FUNCTION_BLOCK VirtualMaster EXTENDS FB_PackML_BaseModule
VAR
	Axis : FB_Component_BasicSlaveAxis := (Name := 'Virtual Master');
END_VAR

METHOD PROTECTED Aborting
//Mode is ignored
CASE SequenceState OF
	0:
		NoStateTasksToComplete := FALSE;

		// Stop Axis
		Axis.Override := 100;
		IF Axis.Stop() OR Axis.Error THEN // This will also GearOut
			SequenceState := SequenceState + 10;
		END_IF

	10:
		IF Axis.Stopped THEN
			SequenceState := SequenceState + 10;
		END_IF

	20: // Disable Axis
		IF Axis.Disable() THEN
			SequenceState := SequenceState + 10;
		END_IF

	30:
		IF NOT Axis.Enabled THEN
			SequenceState := SequenceState + 10;
		END_IF

	40:
		StateTasksComplete := TRUE;
END_CASE

SUPER^.Aborting();
END_METHOD

PROPERTY AxisRef : REFERENCE TO AXIS_REF
GET
AxisRef REF= Axis.Axis;
END_GET
END_PROPERTY

METHOD PROTECTED Completing
CASE _CurrentMode OF
	ePMLUnitMode_Production:
		CASE SequenceState OF
			0:
				NoStateTasksToComplete := FALSE;
				IF Axis.Stop() THEN
					SequenceState := SequenceState + 10;
				END_IF

			10:
				IF Axis.Stopped THEN
					SequenceState := SequenceState + 10;
				END_IF

			20:
				StateTasksComplete := TRUE;
		END_CASE

	ePMLProtUnitMode_Maintenance, ePMLProtUnitMode_Manual:
		;
END_CASE

SUPER^.Completing();
END_METHOD

METHOD PUBLIC CyclicLogic
IF NOT InitComplete THEN
	_InitComplete := Initialize();
	RETURN;
END_IF

SUPER^.CyclicLogic();
END_METHOD

METHOD PROTECTED Initialize : BOOL;
Initialize := FALSE;
CASE DescendantSequenceState OF
	0:
		RegisterComponent(Axis);
		DescendantSequenceState := DescendantSequenceState + 10;

	10:
		IF SUPER^.Initialize() THEN
			DescendantSequenceState := DescendantSequenceState + 10;
		END_IF

	20:
		Initialize := TRUE;
END_CASE
END_METHOD

METHOD PROTECTED Starting
CASE _CommandedMode OF
	ePMLProtUnitMode_Production:
		CASE SequenceState OF
			0:
				NoStateTasksToComplete := FALSE;
				IF Axis.Enable() THEN
					SequenceState := SequenceState + 10;
				END_IF

			10:
				IF Axis.Enabled THEN
					SequenceState := SequenceState + 10;
				END_IF

			20:
				StateTasksComplete := TRUE;
		END_CASE
END_CASE

SUPER^.Starting();
END_METHOD

METHOD PROTECTED Stopping
CASE _CurrentMode OF
	ePMLUnitMode_Production:
		CASE SequenceState OF
			0:
				NoStateTasksToComplete := FALSE;
				IF Axis.Stop() THEN //This will also GearOut
					SequenceState := SequenceState + 10;
				END_IF

			10:
				IF Axis.Stopped THEN
					SequenceState := SequenceState + 10;
				END_IF

			20:
				StateTasksComplete := TRUE;
		END_CASE
END_CASE

SUPER^.Stopping();
END_METHOD

END_FUNCTION_BLOCK

(* stored: Version 1.1.0.1, ProductVersion 3.1.4024.12
   POU VirtualMaster: Id {e8eb8946-ac6b-4f9a-a349-a2038fff9f99}, SpecialFunc None
   Folder Acting States: Id {0e7fcdd1-1a47-47b7-afb6-15dec58e89f0}
   Folder CyclicLogic: Id {9507ba62-34dd-4882-8303-6629ec3ae7d0}
   Folder Initialize: Id {dd24a89b-da86-48b0-a283-f4387229524d}
   Method Aborting: Id {0ab2a755-f479-4155-bea8-7b1b108018b5}
   Property AxisRef: Id {8fbb3c08-11e6-42e9-be14-c11d172359bb}
   Get Get: Id {2a15330a-5ee0-4def-aebb-a9f06cee8655}
   Method Completing: Id {3ff898da-49a5-42a9-84dc-dd8eaed69c93}
   Method CyclicLogic: Id {099d02ae-52c4-4630-a76e-d553625d2bca}
   Method Initialize: Id {6642d997-98c2-45af-8731-ca9c93da577c}
   Method Starting: Id {d700bbd5-4ebd-42aa-9db1-b591835e231d}
   Method Stopping: Id {1d286d67-4c20-4caf-b756-9a8f72182cf7} *)
